FUNCTION_BLOCK FB_FieldCodecDouble IMPLEMENTS I_FieldCodec
VAR_INPUT
END_VAR
VAR_OUTPUT
END_VAR
VAR
    fValue : LREAL;
END_VAR

METHOD CalculatePackedDataSize : HRESULT
VAR_INPUT CONSTANT
	anyFirstElem	: T_Any;
	nLength	        : UDINT;        // items to write
END_VAR
VAR_OUTPUT
    nPackedDataSize : UDINT;
END_VAR
VAR
    anyItem         : T_ANY;
    i               : UDINT;
    fValue          : LREAL;
END_VAR
anyItem := anyFirstElem;

IF nLength < 1 THEN
    nPackedDataSize := 0;
    RETURN;
END_IF

FOR i := 0  TO nLength - 1 DO
    anyItem.pValue := anyFirstElem.pValue + (i * TO_UDINT(anyFirstElem.diSize)); 
    fValue := PLREAL_TO_LREAL(anyItem.pValue);
    nPackedDataSize := nPackedDataSize + F_ComputeDoubleSize(fValue);
END_FOR
END_METHOD

METHOD IsPackedRepeatedField : BOOL
VAR_INPUT
	nTag	: UDINT;
END_VAR
IsPackedRepeatedField := F_IsPackedRepeatedField(nTag);
END_METHOD


METHOD ValueReader : HRESULT
VAR_IN_OUT
    stBuffer : ST_Span;
	stState	: ST_ParserInternalState;
END_VAR
VAR_OUTPUT
	anyOut	: T_Any;
END_VAR

ValueReader := F_ParseDouble(stBuffer, stState, fValue=> fValue);
anyOut := F_ToAnyType(anyArg:= fValue);
END_METHOD

METHOD ValueWriter : HRESULT
VAR_IN_OUT
    stBuffer : ST_Span;
    stState  : ST_WriterInternalState;
END_VAR
VAR_INPUT
    anyIn : T_ANY;
END_VAR
VAR
    fValue  : LREAL;
END_VAR

fValue := PLREAL_TO_LREAL(anyIn.pValue);
ValueWriter := F_WriteDouble(stBuffer, stState, fValue);
END_METHOD

END_FUNCTION_BLOCK

(* stored: Version 1.1.0.1
   POU FB_FieldCodecDouble: Id {f6635256-2255-4dad-ac3d-fde3245c6d0d}, SpecialFunc None
   Method CalculatePackedDataSize: Id {ef2a42bf-2f87-4692-a9f3-567b05e779b1}
   Method IsPackedRepeatedField: Id {d9206b81-f1d0-4f9c-8b27-a7557037cb20}
   Method ValueReader: Id {47db2cd1-e3bd-4ae3-8d15-00da42a68236}
   Method ValueWriter: Id {4ed72eef-3be8-496d-a27c-b8015cf6d975} *)
